// TIA Portal V18 export
VAR_GLOBAL   // PLC tag table "CentralShifter"
   iCS_SensorHoming_Left AT %I800.0 : Bool;
   iCS_SensorHoming_Right AT %I800.1 : Bool;
END_VAR
